// TIA Portal V20 export
DATA_BLOCK "GDB_PalletizingPath"   // DB15
TITLE = Palletizing buffered-path command list (V4.0)
{ S7_Optimized_Access := 'TRUE' }
// Buffered-path command list for the V4.0 palletizing executor. Array of UDT_PathCmd, built once per bo_InitPallet rising edge and executed by FB_AutoCtrl_Palletizing REGION 4. Kept as a separate global DB (not an instance-DB stat array) so the PowerShell smoke harness can probe aCmd[n] directly.
// stored: MemoryReserve 100
   VAR
      aCmd : Array[1..200] of "UDT_PathCmd";   // Buffered-path command list -- built by FB_AutoCtrl_Palletizing REGION 1 (9 commands per box x 16 boxes + 1 END_OF_PATH ~= 145 used) and walked by the REGION 4 executor. [1..200] gives headroom.
      i16_CmdCount : Int;   // Number of valid commands in aCmd, set by REGION 1 after building the list. The END_OF_PATH command sits at aCmd[i16_CmdCount].
   END_VAR
BEGIN
END_DATA_BLOCK
